FUNCTION_BLOCK FB_ReceivegdTemp_Right
VAR_IN_OUT
	Inputs_Right : CANRXQUEUESTRUCT_E_32;
	Outputs_Right : CANTXQUEUESTRUCT_E_32;
END_VAR
VAR_OUTPUT
	Temp_a_gd_Right : LREAL;
	Temp_b_gd_Right : LREAL;
	Temp_c_gd_Right : LREAL;
END_VAR
VAR
	MessageReceived : ARRAY[0..31] OF EXTCANQUEUE;
	i : INT;
	
	fbPPS_Timer : TON;
	nPacketsPerSecond: INT;
	nReceiveCounter : INT;
	nLastReceiveCounter : INT;
END_VAR

FOR i := 0 TO (Inputs_Right.NoOfRxMessages-1) DO
    IF Inputs_Right.RxMessages[i].cobId = 700 THEN 
        Temp_a_gd_Right := INT_TO_LREAL(WORD_TO_INT(SHL(USINT_TO_UINT(Inputs_Right.RxMessages[i].data[0]), 8) OR USINT_TO_UINT(Inputs_Right.RxMessages[i].data[1]))) / 10.0; 
        Temp_b_gd_Right := INT_TO_LREAL(WORD_TO_INT(SHL(USINT_TO_UINT(Inputs_Right.RxMessages[i].data[2]), 8) OR USINT_TO_UINT(Inputs_Right.RxMessages[i].data[3]))) / 10.0; 
        Temp_c_gd_Right := INT_TO_LREAL(WORD_TO_INT(SHL(USINT_TO_UINT(Inputs_Right.RxMessages[i].data[4]), 8) OR USINT_TO_UINT(Inputs_Right.RxMessages[i].data[5]))) / 10.0;
		nReceiveCounter := nReceiveCounter + 1; 
    END_IF
END_FOR
fbPPS_Timer(IN := NOT fbPPS_Timer.Q, PT := T#1S);
IF fbPPS_Timer.Q THEN
			nPacketsPerSecond   := nReceiveCounter - nLastReceiveCounter;
			nLastReceiveCounter := nReceiveCounter;
END_IF

END_FUNCTION_BLOCK

(* stored: Version 1.1.0.1
   POU FB_ReceivegdTemp_Right: Id {958e701c-fb98-4994-9586-25692d9df0a7}, SpecialFunc None *)
